// TIA Portal V19 export
TYPE "Positioning_EPOS_Machine_COut"
// stored: Access Published
   STRUCT
      Infeed_ReqON : Bool;
      CtrlSafe : Bool;
      Homed : Bool;   // Axis is homed
      Standstill : Bool;
      Enabled : Bool;   // Axis power is on (drive enabled)
      InPosition : Bool;
      MinusCheckNext : Bool;
      PlusCheckNext : Bool;
      MinusRunning : Bool;
      PlusRunning : Bool;
      MinusLsSwReached : Bool;
      PlusLsSwReached : Bool;
      MinusLimitReached : Bool;
      PlusLimitReached : Bool;
      ActualPosition : LReal;
      ActualTargetPos : LReal;
      MinPosition : LReal;
      MaxPosition : LReal;
      ActualVelocity : LReal;
      MaxVelocity : LReal;
   END_STRUCT;
END_TYPE
